{attribute 'GeneratedUsingTerminal: EL9576-0000-0022'}
{attribute addProperty BoxType "EL9576-0000-0022"}
{attribute addProperty Id "Terminal_OvertemperatureAT %I*BOOL1I2T_errorAT %I*BOOL1I2T_warningAT %I*BOOL1OvervoltageAT %I*BOOL1UndervoltageAT %I*BOOL1Chopper_onAT %I*BOOL1Overcurrent_ProtectionAT %I*BOOL1Input_cycle_counterAT %I*BYTE1DC_link_voltageAT %I*UDINT4Resistor_CurrentAT %I*DINT4Duty_CycleAT %I*USINT1"}
{attribute addProperty CRC "2060357542"}
{attribute addProperty Size "17"}
TYPE BCT_Inputs_7ACE8FA6 EXTENDS InputBase_8311D824 :
STRUCT
	{attribute addProperty Name "Terminal_Overtemperature"}
	Terminal_Overtemperature AT %I* : BOOL;
	{attribute addProperty Name "I2T_error"}
	I2T_error AT %I* : BOOL;
	{attribute addProperty Name "I2T_warning"}
	I2T_warning AT %I* : BOOL;
	{attribute addProperty Name "Overvoltage"}
	Overvoltage AT %I* : BOOL;
	{attribute addProperty Name "Undervoltage"}
	Undervoltage AT %I* : BOOL;
	{attribute addProperty Name "Chopper_on"}
	Chopper_on AT %I* : BOOL;
	{attribute addProperty Name "Overcurrent_Protection"}
	Overcurrent_Protection AT %I* : BOOL;
	{attribute addProperty Name "Input_cycle_counter"}
	Input_cycle_counter AT %I* : BYTE;
	{attribute addProperty Name "DC_link_voltage"}
	DC_link_voltage AT %I* : UDINT;
	{attribute addProperty Name "Resistor_Current"}
	Resistor_Current AT %I* : DINT;
	{attribute addProperty Name "Duty_Cycle"}
	Duty_Cycle AT %I* : USINT;
END_STRUCT
END_TYPE

(* stored: Version 1.2.0.0, ProductVersion 3.1.4024.9
   DUT BCT_Inputs_7ACE8FA6: Id {fb2855b0-1445-412b-b589-14dccd633013} *)
